REGION Network 73: Tracking from Stacker to Shuttle
   #_w1 := ("BTrk".A0303.Stacker.Completato OR (("BTrk".A0303.Stacker.Layers_Qty >= "BTrk".A0303.Stacker.Layers_Target) AND ("BTrk".A0303.Stacker.Layers_Target <> 0))) AND #SollevatoreCodaInPosDeposito AND #SollevatoreTestaInPosDeposito AND #CIn.Navetta.ReadyToRecive AND "BTrk".A0304.Empty;
   #PE.TrkToShuttle := #_w1 AND NOT #AUX.TrkToShuttle;   // rising edge
   #AUX.TrkToShuttle := #_w1;
   IF #PE.TrkToShuttle THEN
       "BTrk".A0304.Layers := "BTrk".A0303.Stacker.Layers;
       "BTrk".A0303.Stacker.Layers := "BTrk".EmptyLayers;
   END_IF;
END_REGION

REGION Network 75: <<< OP CAN MOVE FREELY >>>
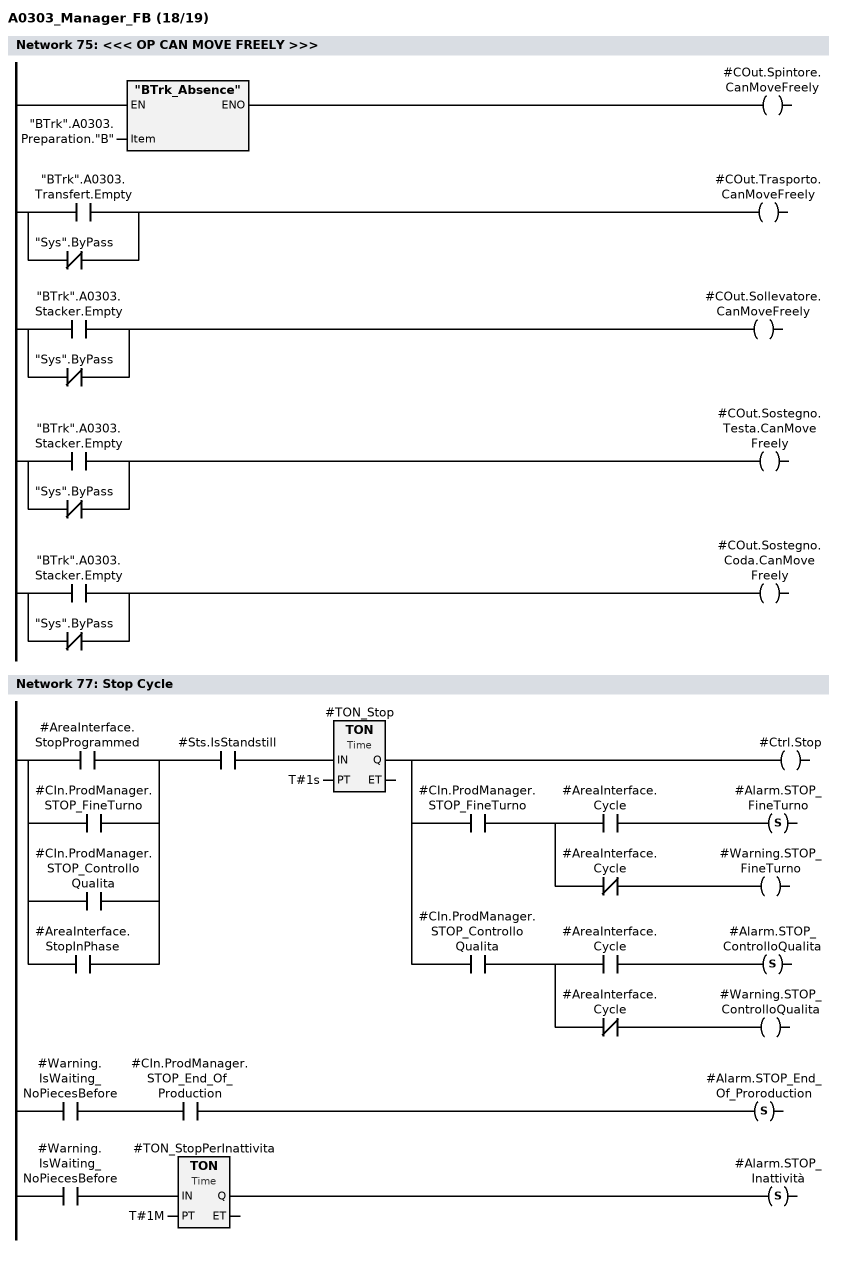
   RUNG wire#powerrail
      "BTrk_Absence"(Item := "BTrk".A0303.Preparation."B")
      Coil( #COut.Spintore.CanMoveFreely )
   END_RUNG
   RUNG wire#powerrail
      Contact( "BTrk".A0303.Transfert.Empty )
      wire#w1
      Coil( #COut.Trasporto.CanMoveFreely )
   END_RUNG
   RUNG wire#powerrail
      I_Contact( "Sys".ByPass )
   END_RUNG wire#w1
   RUNG wire#powerrail
      Contact( "BTrk".A0303.Stacker.Empty )
      wire#w2
      Coil( #COut.Sollevatore.CanMoveFreely )
   END_RUNG
   RUNG wire#powerrail
      I_Contact( "Sys".ByPass )
   END_RUNG wire#w2
   RUNG wire#powerrail
      Contact( "BTrk".A0303.Stacker.Empty )
      wire#w3
      Coil( #COut.Sostegno.Testa.CanMoveFreely )
   END_RUNG
   RUNG wire#powerrail
      I_Contact( "Sys".ByPass )
   END_RUNG wire#w3
   RUNG wire#powerrail
      Contact( "BTrk".A0303.Stacker.Empty )
      wire#w4
      Coil( #COut.Sostegno.Coda.CanMoveFreely )
   END_RUNG
   RUNG wire#powerrail
      I_Contact( "Sys".ByPass )
   END_RUNG wire#w4
   // the same network as SCL:
   "BTrk_Absence"(Item := "BTrk".A0303.Preparation."B", ENO => #_w1);
   #COut.Spintore.CanMoveFreely := #_w1;
   #COut.Trasporto.CanMoveFreely := "BTrk".A0303.Transfert.Empty OR NOT "Sys".ByPass;
   #COut.Sollevatore.CanMoveFreely := "BTrk".A0303.Stacker.Empty OR NOT "Sys".ByPass;
   #COut.Sostegno.Testa.CanMoveFreely := "BTrk".A0303.Stacker.Empty OR NOT "Sys".ByPass;
   #COut.Sostegno.Coda.CanMoveFreely := "BTrk".A0303.Stacker.Empty OR NOT "Sys".ByPass;
END_REGION

REGION Network 77: Stop Cycle
   RUNG wire#powerrail
      Contact( #AreaInterface.StopProgrammed )
      wire#w1
      Contact( #Sts.IsStandstill )
      { S7_Templates := "time_type := Time" } #TON_Stop.TON(pt := T#1s, et =>)
      wire#w2
      Coil( #Ctrl.Stop )
   END_RUNG
   RUNG wire#powerrail
      Contact( #CIn.ProdManager.STOP_FineTurno )
   END_RUNG wire#w1
   RUNG wire#powerrail
      Contact( #CIn.ProdManager.STOP_ControlloQualita )
   END_RUNG wire#w1
   RUNG wire#powerrail
      Contact( #AreaInterface.StopInPhase )
   END_RUNG wire#w1
   RUNG wire#w2
      Contact( #CIn.ProdManager.STOP_FineTurno )
      wire#w3
      Contact( #AreaInterface.Cycle )
      S_Coil( #Alarm.STOP_FineTurno )
   END_RUNG
   RUNG wire#w3
      I_Contact( #AreaInterface.Cycle )
      Coil( #Warning.STOP_FineTurno )
   END_RUNG
   RUNG wire#w2
      Contact( #CIn.ProdManager.STOP_ControlloQualita )
      wire#w4
      Contact( #AreaInterface.Cycle )
      S_Coil( #Alarm.STOP_ControlloQualita )
   END_RUNG
   RUNG wire#w4
      I_Contact( #AreaInterface.Cycle )
      Coil( #Warning.STOP_ControlloQualita )
   END_RUNG
   RUNG wire#powerrail
      Contact( #Warning.IsWaiting_NoPiecesBefore )
      Contact( #CIn.ProdManager.STOP_End_Of_Production )
      S_Coil( #Alarm.STOP_End_Of_Proroduction )
   END_RUNG
   RUNG wire#powerrail
      Contact( #Warning.IsWaiting_NoPiecesBefore )
      { S7_Templates := "time_type := Time" } #TON_StopPerInattivita.TON(pt := T#1M, et =>)
      S_Coil( #Alarm.STOP_Inattività )
   END_RUNG
   // the same network as SCL:
   #TON_Stop.TON(IN := (#AreaInterface.StopProgrammed OR #CIn.ProdManager.STOP_FineTurno OR #CIn.ProdManager.STOP_ControlloQualita OR #AreaInterface.StopInPhase) AND #Sts.IsStandstill,
                 PT := T#1s);
   #Ctrl.Stop := #TON_Stop.Q;
   #_w1 := #TON_Stop.Q AND #CIn.ProdManager.STOP_FineTurno;
   IF #_w1 AND #AreaInterface.Cycle THEN #Alarm.STOP_FineTurno := TRUE; END_IF;
   #Warning.STOP_FineTurno := #_w1 AND NOT #AreaInterface.Cycle;
   #_w2 := #TON_Stop.Q AND #CIn.ProdManager.STOP_ControlloQualita;
   IF #_w2 AND #AreaInterface.Cycle THEN #Alarm.STOP_ControlloQualita := TRUE; END_IF;
   #Warning.STOP_ControlloQualita := #_w2 AND NOT #AreaInterface.Cycle;
   IF #Warning.IsWaiting_NoPiecesBefore AND #CIn.ProdManager.STOP_End_Of_Production THEN
       #Alarm.STOP_End_Of_Proroduction := TRUE;
   END_IF;
   #TON_StopPerInattivita.TON(IN := #Warning.IsWaiting_NoPiecesBefore, PT := T#1M);
   IF #TON_StopPerInattivita.Q THEN #Alarm.STOP_Inattività := TRUE; END_IF;
END_REGION

REGION Network 79 (SCL): SYNOPTIC
END_REGION

REGION Network 80: << FINAL OPERATIONS >>
   // +
   // +
   // +
   // +
   // +
   // +
   // +
   // +
   // +
   // +
   // +
   // +
   // +
END_REGION

REGION Network 81: All motions standstill
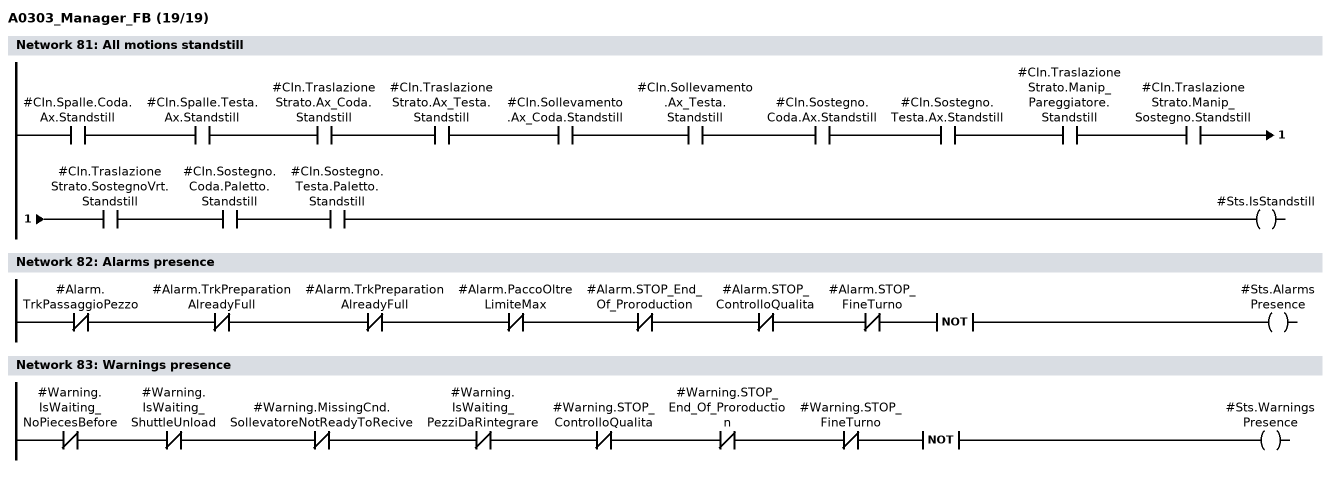
   RUNG wire#powerrail
      Contact( #CIn.Spalle.Coda.Ax.Standstill )
      Contact( #CIn.Spalle.Testa.Ax.Standstill )
      Contact( #CIn.TraslazioneStrato.Ax_Coda.Standstill )
      Contact( #CIn.TraslazioneStrato.Ax_Testa.Standstill )
      Contact( #CIn.Sollevamento.Ax_Coda.Standstill )
      Contact( #CIn.Sollevamento.Ax_Testa.Standstill )
      Contact( #CIn.Sostegno.Coda.Ax.Standstill )
      Contact( #CIn.Sostegno.Testa.Ax.Standstill )
      Contact( #CIn.TraslazioneStrato.Manip_Pareggiatore.Standstill )
      Contact( #CIn.TraslazioneStrato.Manip_Sostegno.Standstill )
      Contact( #CIn.TraslazioneStrato.SostegnoVrt.Standstill )
      Contact( #CIn.Sostegno.Coda.Paletto.Standstill )
      Contact( #CIn.Sostegno.Testa.Paletto.Standstill )
      Coil( #Sts.IsStandstill )
   END_RUNG
   // the same network as SCL:
   #Sts.IsStandstill := #CIn.Spalle.Coda.Ax.Standstill AND #CIn.Spalle.Testa.Ax.Standstill AND #CIn.TraslazioneStrato.Ax_Coda.Standstill AND #CIn.TraslazioneStrato.Ax_Testa.Standstill AND #CIn.Sollevamento.Ax_Coda.Standstill AND #CIn.Sollevamento.Ax_Testa.Standstill AND #CIn.Sostegno.Coda.Ax.Standstill AND #CIn.Sostegno.Testa.Ax.Standstill AND #CIn.TraslazioneStrato.Manip_Pareggiatore.Standstill AND #CIn.TraslazioneStrato.Manip_Sostegno.Standstill AND #CIn.TraslazioneStrato.SostegnoVrt.Standstill AND #CIn.Sostegno.Coda.Paletto.Standstill AND #CIn.Sostegno.Testa.Paletto.Standstill;
END_REGION

REGION Network 82: Alarms presence
   RUNG wire#powerrail
      I_Contact( #Alarm.TrkPassaggioPezzo )
      I_Contact( #Alarm.TrkPreparationAlreadyFull )
      I_Contact( #Alarm.TrkPreparationAlreadyFull )
      I_Contact( #Alarm.PaccoOltreLimiteMax )
      I_Contact( #Alarm.STOP_End_Of_Proroduction )
      I_Contact( #Alarm.STOP_ControlloQualita )
      I_Contact( #Alarm.STOP_FineTurno )
      Not()
      Coil( #Sts.AlarmsPresence )
   END_RUNG
   // the same network as SCL:
   #Sts.AlarmsPresence := NOT (NOT #Alarm.TrkPassaggioPezzo AND NOT #Alarm.TrkPreparationAlreadyFull AND NOT #Alarm.TrkPreparationAlreadyFull AND NOT #Alarm.PaccoOltreLimiteMax AND NOT #Alarm.STOP_End_Of_Proroduction AND NOT #Alarm.STOP_ControlloQualita AND NOT #Alarm.STOP_FineTurno);
END_REGION

REGION Network 83: Warnings presence
   RUNG wire#powerrail
      I_Contact( #Warning.IsWaiting_NoPiecesBefore )
      I_Contact( #Warning.IsWaiting_ShuttleUnload )
      I_Contact( #Warning.MissingCnd.SollevatoreNotReadyToRecive )
      I_Contact( #Warning.IsWaiting_PezziDaRintegrare )
      I_Contact( #Warning.STOP_ControlloQualita )
      I_Contact( #Warning.STOP_End_Of_Proroduction )
      I_Contact( #Warning.STOP_FineTurno )
      Not()
      Coil( #Sts.WarningsPresence )
   END_RUNG
   // the same network as SCL:
   #Sts.WarningsPresence := NOT (NOT #Warning.IsWaiting_NoPiecesBefore AND NOT #Warning.IsWaiting_ShuttleUnload AND NOT #Warning.MissingCnd.SollevatoreNotReadyToRecive AND NOT #Warning.IsWaiting_PezziDaRintegrare AND NOT #Warning.STOP_ControlloQualita AND NOT #Warning.STOP_End_Of_Proroduction AND NOT #Warning.STOP_FineTurno);
END_REGION

REGION Network 84 (SCL): Collect machine to area interface
   #MachineInterface.AlarmsPresence := #Sts.AlarmsPresence;

   #MachineInterface.WarningPresence := #Sts.WarningsPresence;

   #MachineInterface.MotionsStandStill := #Sts.IsStandstill;

   #MachineInterface.AutReady := #AreaInterface.Aut AND NOT #Sts.AlarmsPresence;


   #MachineInterface.AckStopInPhase := #AreaInterface.StopInPhase AND #Ctrl.Stop;

   #MachineInterface.AckStopProgrammed := #AreaInterface.StopProgrammed AND #Ctrl.Stop;


   #MachineInterface.Aborting := #AreaInterface.Aut AND #Sts.AlarmsPresence;
END_REGION
END_FUNCTION_BLOCK
